(* IEC 61131-3 sources: POMIRTS_lab3/AS/Library/AsNxDnM, 3 files *)

(* ---- AsNxDnM.typ ---- *)
(********************************************************************
 * COPYRIGHT -- Bernecker + Rainer
 ********************************************************************
 * Library: AsNxDnM
 * File: AsNxDnM.typ
 * Author: B+R
 ********************************************************************
 * Data types of library AsNxDnM
 ********************************************************************)

TYPE
	nxdnmSlaveList_t		: STRUCT			(*slave list*)
		slave				: ARRAY[0..63] OF BOOL;
	END_STRUCT;

	nxdnmLifeList_t			: STRUCT			(*life list*)
		slave				: ARRAY[0..63] OF USINT;
	END_STRUCT;

	nxdnmDiagData_t			: STRUCT			(*diagnostic data*)
		nodeExtraDiag		: USINT;
		devMainState		: USINT;
		onlineError			: USINT;
		generalErrorCode	: USINT;
		additionalCode		: USINT;
		heartBeatTimeout	: UINT;
	END_STRUCT;

	nxdnmResData_t			: STRUCT			(*response data*)
		macId				: USINT;
		length				: USINT;
		data				: ARRAY[0..7] OF USINT;
	END_STRUCT;

	nxdnmResDataList_t		: STRUCT			(*response data list*)
		slave				: ARRAY[0..63] OF nxdnmResData_t;
	END_STRUCT;
END_TYPE

(* ---- AsNxDnM.fun ---- *)
(********************************************************************
 * COPYRIGHT -- Bernecker + Rainer
 ********************************************************************
 * Library: AsNxDnM
 * File: AsNxDnM.fun
 * Author: B+R
 ********************************************************************
 * Functions and function blocks of library AsNxDnM
 ********************************************************************)

FUNCTION_BLOCK nxdnmSetOperationMode	(*set operation mode*)
	VAR_INPUT
		enable			: BOOL;			(*enables execution*)
		pDevice			: UDINT;		(*interface name given as a pointer, e.g., "SL<x>.SS<y>.IF<z>"*)
		mode			: UDINT;		(*operation mode*)
	END_VAR
	VAR
        _state			: UINT;			(*internal variable*)
		_result			: UINT;			(*internal variable*)
        _srcId			: UDINT;		(*internal variable*)
	END_VAR
	VAR_OUTPUT
		status			: UINT;			(*execution status: ERR_OK, ERR_FUB_ENABLE_FALSE, ERR_FUB_BUSY, 0xXXXX = see help*)
		dnStatus		: UDINT;		(*devicenet stack status*)
	END_VAR
END_FUNCTION_BLOCK

FUNCTION_BLOCK nxdnmGetAttribute		(*get attribute*)
	VAR_INPUT
		enable			: BOOL;			(*enables execution*)
		pDevice			: UDINT;		(*interface name given as a pointer, e.g., "SL<x>.SS<y>.IF<z>"*)
		macId			: USINT;		(*device mac id*)
		classId			: UINT;			(*class id*)
		instanceId		: UINT;			(*instance id*)
		attributeId		: UINT;			(*attribute id*)
		attLengthMax	: UINT;			(*maximum attribute data length*)
		pAttData		: UDINT;		(*attribute data given as pointer*)
	END_VAR
	VAR
        _state			: UINT;			(*internal variable*)
		_result			: UINT;			(*internal variable*)
        _srcId			: UDINT;		(*internal variable*)
	END_VAR
	VAR_OUTPUT
		status			: UINT;			(*execution status: ERR_OK, ERR_FUB_ENABLE_FALSE, ERR_FUB_BUSY, 0xXXXX = see help*)
		dnStatus		: UDINT;		(*devicenet stack status*)
		attLength		: UINT;			(*attribute data length*)
		generalError	: USINT;		(*general error*)
		additionalError	: USINT;		(*additional error*)
	END_VAR
END_FUNCTION_BLOCK

FUNCTION_BLOCK nxdnmSetAttribute		(*set attribute*)
	VAR_INPUT
		enable			: BOOL;			(*enables execution*)
		pDevice			: UDINT;		(*interface name given as a pointer, e.g., "SL<x>.SS<y>.IF<z>"*)
		macId			: USINT;		(*device mac id*)
		classId			: UINT;			(*class id*)
		instanceId		: UINT;			(*instance id*)
		attributeId		: UINT;			(*attribute id*)
		attLength		: UINT;			(*attribute data length*)
		pAttData		: UDINT;		(*attribute data given as pointer*)
	END_VAR
	VAR
        _state			: UINT;			(*internal variable*)
		_result			: UINT;			(*internal variable*)
        _srcId			: UDINT;		(*internal variable*)
	END_VAR
	VAR_OUTPUT
		status			: UINT;			(*execution status: ERR_OK, ERR_FUB_ENABLE_FALSE, ERR_FUB_BUSY, 0xXXXX = see help*)
		dnStatus		: UDINT;		(*devicenet stack status*)
		generalError	: USINT;		(*general error*)
		additionalError	: USINT;		(*additional error*)
	END_VAR
END_FUNCTION_BLOCK

FUNCTION_BLOCK nxdnmAcyclicBitStrobing	(*acyclic bit strobing*)
	VAR_INPUT
		enable			: BOOL;			(*enables execution*)
		pDevice			: UDINT;		(*interface name given as a pointer, e.g., "SL<x>.SS<y>.IF<z>"*)
		pStrobeMask		: UDINT;		(*strobe mask given as pointer*)
		pStrobeCommand	: UDINT;		(*strobe command given as pointer*)
		pStatusList		: UDINT;		(*status list given as pointer*)
		pResDataList	: UDINT;		(*response data list given as pointer*)
		timeout			: UDINT;		(*timeout*)
	END_VAR
	VAR
        _state			: UINT;			(*internal variable*)
		_result			: UINT;			(*internal variable*)
        _srcId			: UDINT;		(*internal variable*)
	END_VAR
	VAR_OUTPUT
		status			: UINT;			(*execution status: ERR_OK, ERR_FUB_ENABLE_FALSE, ERR_FUB_BUSY, 0xXXXX = see help*)
		dnStatus		: UDINT;		(*devicenet stack status*)
	END_VAR
END_FUNCTION_BLOCK

FUNCTION_BLOCK nxdnmLifeList			(*life list*)
	VAR_INPUT
		enable			: BOOL;			(*enables execution*)
		pDevice			: UDINT;		(*interface name given as a pointer, e.g., "SL<x>.SS<y>.IF<z>"*)
		timeout			: UDINT;		(*timeout*)
		pLifeList		: UDINT;		(*life list given as pointer*)
	END_VAR
	VAR
        _state			: UINT;			(*internal variable*)
		_result			: UINT;			(*internal variable*)
        _srcId			: UDINT;		(*internal variable*)
	END_VAR
	VAR_OUTPUT
		status			: UINT;			(*execution status: ERR_OK, ERR_FUB_ENABLE_FALSE, ERR_FUB_BUSY, 0xXXXX = see help*)
		dnStatus		: UDINT;		(*devicenet stack status*)
	END_VAR
END_FUNCTION_BLOCK

FUNCTION_BLOCK nxdnmDiagnostics			(*diagnostics*)
	VAR_INPUT
		enable			: BOOL;			(*enables execution*)
		pDevice			: UDINT;		(*interface name given as a pointer, e.g., "SL<x>.SS<y>.IF<z>"*)
		macId			: USINT;		(*device mac id*)
		getOnly			: BOOL;			(*get only flag*)
		diagLengthMax	: UDINT;		(*maximum diagnostic data length*)
		pDiagData		: UDINT;		(*diagnostic data given as pointer*)
	END_VAR
	VAR
        _state			: UINT;			(*internal variable*)
		_result			: UINT;			(*internal variable*)
        _srcId			: UDINT;		(*internal variable*)
	END_VAR
	VAR_OUTPUT
		status			: UINT;			(*execution status: ERR_OK, ERR_FUB_ENABLE_FALSE, ERR_FUB_BUSY, 0xXXXX = see help*)
		dnStatus		: UDINT;		(*devicenet stack status*)
		diagLength		: UDINT;		(*diagonstic data length*)
	END_VAR
END_FUNCTION_BLOCK

(* ---- AsNxDnM.var ---- *)
(********************************************************************
 * COPYRIGHT -- Bernecker + Rainer
 ********************************************************************
 * Library: AsNxDnM
 * File: AsNxDnM.var
 * Author: B+R
 ********************************************************************
 * Local variables of library AsNxDnM
 ********************************************************************)

VAR CONSTANT
	nxdnmERR_INVALID_DEVICE					: UINT	:= 35380;		(*error invalid device*)
	nxdnmERR_SEND_MESSAGE					: UINT	:= 35381;		(*error send message*)
	nxdnmERR_TIMEOUT						: UINT	:= 35382;		(*error timeout*)
	nxdnmERR_DEVICENET_STACK				: UINT	:= 35383;		(*error receive message*)
	nxdnmERR_PARAMETER						: UINT	:= 35384;		(*error invalid parameter*)
	nxdnmERR_DATALEN						: UINT	:= 35385;		(*error data length*)

	nxdnmFAL_MODE_OFFLINE					: UDINT	:= 16#00;		(*fieldbus application layer mode offline*)
	nxdnmFAL_MODE_STOP						: UDINT	:= 16#40;		(*fieldbus application layer mode stop*)
	nxdnmFAL_MODE_IDLE						: UDINT	:= 16#80;		(*fieldbus application layer mode idle*)
	nxdnmFAL_MODE_RUN						: UDINT	:= 16#C0;		(*fieldbus application layer mode run*)

	nxdnmLIFELIST_OWN_MAC					: USINT	:= 16#FF;		(*responds with own MAC-ID*)
	nxdnmLIFELIST_MAC						: USINT	:= 16#01;		(*responds with MAC-ID*)
	nxdnmLIFELIST_NO_MAC					: USINT	:= 16#00;		(*does not response*)
END_VAR
